FUNCTION_BLOCK CL_AxisMCL2RightBack EXTENDS CL_AxisMC
VAR
  objAxisDriver : CL_AxisDriverL2RightBack;
END_VAR

SUPER^();

METHOD PUBLIC Init : BOOL
VAR_INPUT
  stIrrLine       : ST_LineReference;
  stAxisMotor_P	  : POINTER TO AXIS_REF;
  stAxisMaster_P  : POINTER TO AXIS_REF;
  stDriver        : POINTER TO ST_DriverAX8206_HWI;
END_VAR
Init := FALSE;
IF stDriver <> 0 THEN
  Init := objAxisDriver.Init(stDriver := stDriver);
  Init := Init AND SUPER^.InitMC(stIrrLine := stIrrLine, stAxisMotor_P := stAxisMotor_P, stAxisMaster_P := stAxisMaster_P, AxisDriver_P := ADR(objAxisDriver));
END_IF
END_METHOD

METHOD PROTECTED InitDefect : BOOL
InitDefect := SUPER^.InitDefect();
ADSLOGSTR(ADSLOG_MSGTYPE_LOG, 'CL_AxisMCL2RightBack init defect','');
END_METHOD

METHOD PROTECTED InitParams : BOOL
VAR_INPUT
END_VAR
InitParams := SUPER^.InitParams();
_sWhichAxis := 'right(L2)-back';
_lrInverse := -1.0;
END_METHOD

END_FUNCTION_BLOCK

(* stored: Version 1.1.0.1, ProductVersion 3.1.4024.12
   POU CL_AxisMCL2RightBack: Id {9581f397-500f-4bc2-83c1-3fff25c338cc}, SpecialFunc None
   Method Init: Id {7be38d4e-bda4-4895-b647-4ea29b8b720d}
   Method InitDefect: Id {255aed50-cbe1-4d37-a724-ff92b8ae219e}
   Method InitParams: Id {f630f93c-65da-4341-ab5f-5ba2af850e86} *)
